(* PLC project Unnamed, Unknown Unnamed 1 *)
(* stored: creationDateTime 2025-05-12T19:02:38, modificationDateTime 2025-05-14T16:42:28 *)

PROGRAM traffic
  VAR
    pedestrianButton AT %IX0.0 : BOOL;
    systemButton0 AT %IX0.1 : BOOL;
    pR AT %QX0.4 : BOOL;
    pY AT %QX0.3 : BOOL;
    pG AT %QX0.2 : BOOL;
    cR AT %QX0.7 : BOOL;
    cY AT %QX0.6 : BOOL;
    cG AT %QX0.5 : BOOL;
  END_VAR
  VAR
    TOF0 : TOF;
    SR0 : SR;
    TOF1 : TOF;
    TOF3 : TOF;
    TOF2 : TOF;
    TOF5 : TOF;
    TOF6 : TOF;
  END_VAR
  VAR  (* added by the conversion: wires and edge detectors of the diagram *)
    R_TRIG1 : R_TRIG;
    F_TRIG2 : F_TRIG;
    F_TRIG3 : F_TRIG;
    F_TRIG4 : F_TRIG;
    R_TRIG5 : R_TRIG;
    F_TRIG6 : F_TRIG;
    R_TRIG7 : R_TRIG;
    F_TRIG8 : F_TRIG;
    F_TRIG9 : F_TRIG;
    _XOR52_OUT : BOOL;
  END_VAR

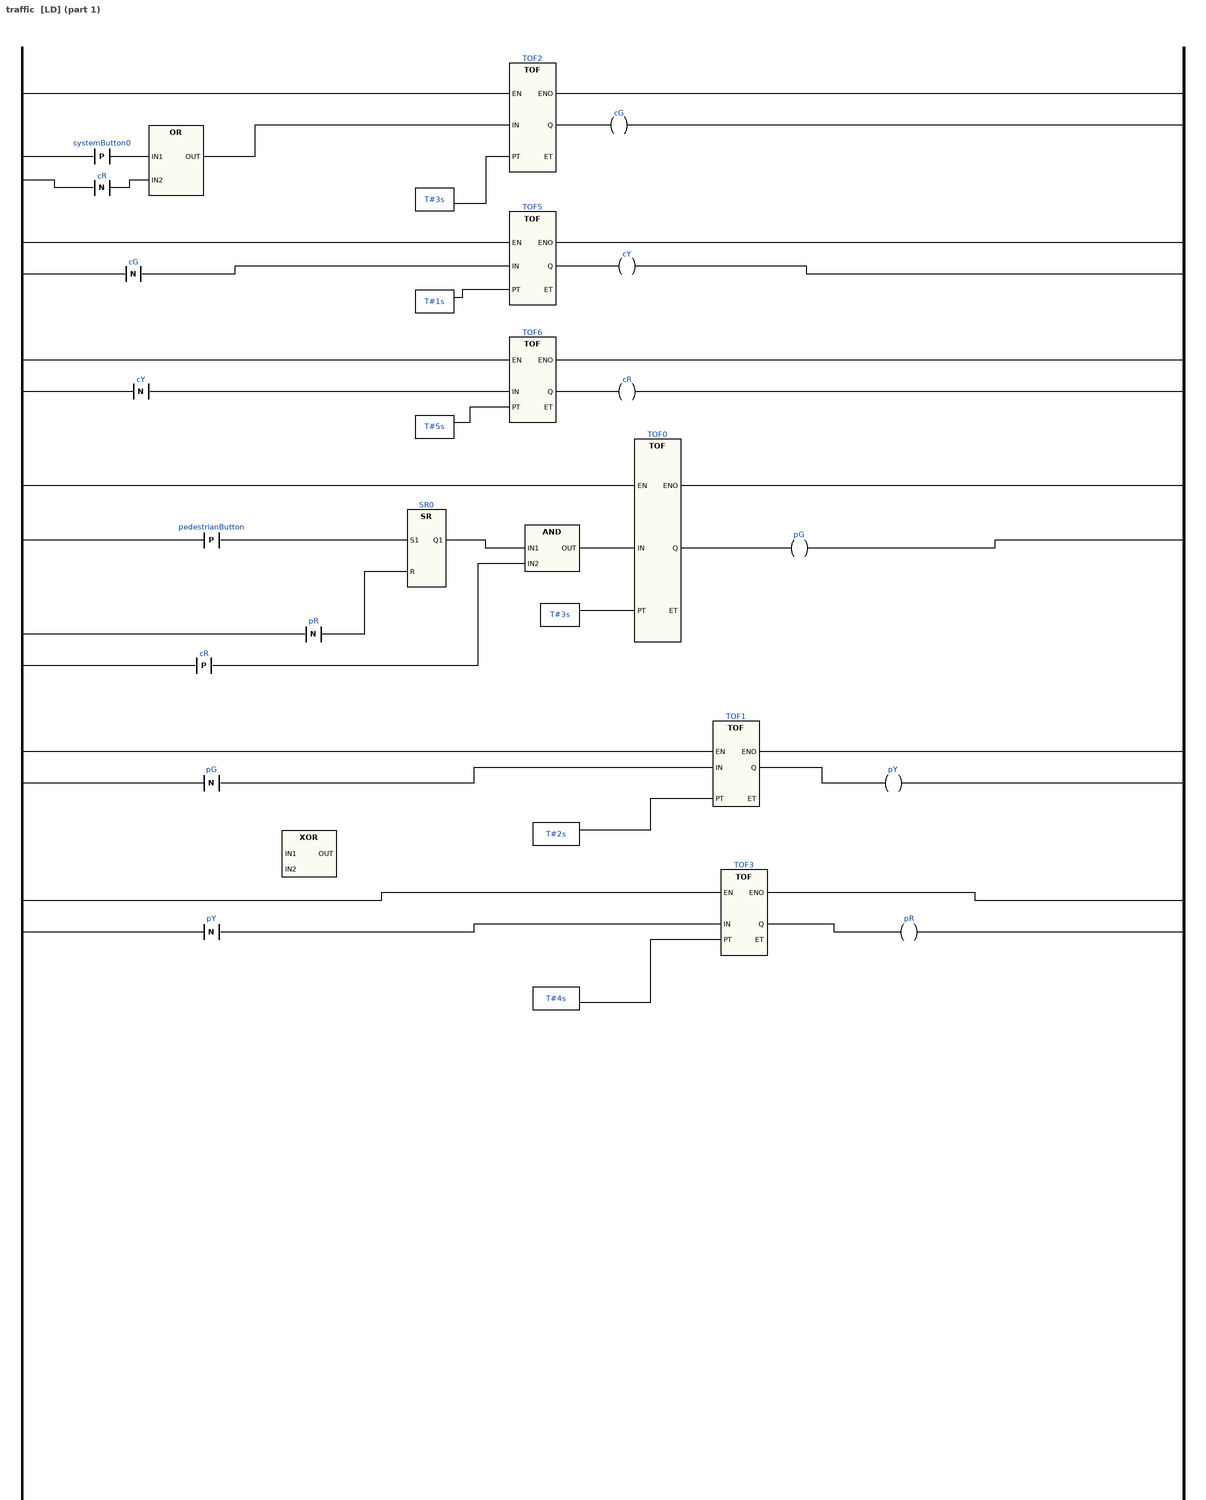
(* LD diagram, written out as Structured Text *)
R_TRIG1(CLK := systemButton0);
F_TRIG2(CLK := cR);
TOF2(IN := R_TRIG1.Q OR F_TRIG2.Q, PT := T#3s);
cG := TOF2.Q;
F_TRIG3(CLK := cG);
TOF5(IN := F_TRIG3.Q, PT := T#1s);
cY := TOF5.Q;
F_TRIG4(CLK := cY);
TOF6(IN := F_TRIG4.Q, PT := T#5s);
cR := TOF6.Q;
R_TRIG5(CLK := pedestrianButton);
F_TRIG6(CLK := pR);
SR0(S1 := R_TRIG5.Q, R := F_TRIG6.Q);
R_TRIG7(CLK := cR);
TOF0(IN := SR0.Q1 AND R_TRIG7.Q, PT := T#3s);
pG := TOF0.Q;
F_TRIG8(CLK := pG);
TOF1(IN := F_TRIG8.Q, PT := T#2s);
pY := TOF1.Q;
F_TRIG9(CLK := pY);
TOF3(IN := F_TRIG9.Q, PT := T#4s);
pR := TOF3.Q;
_XOR52_OUT := XOR();
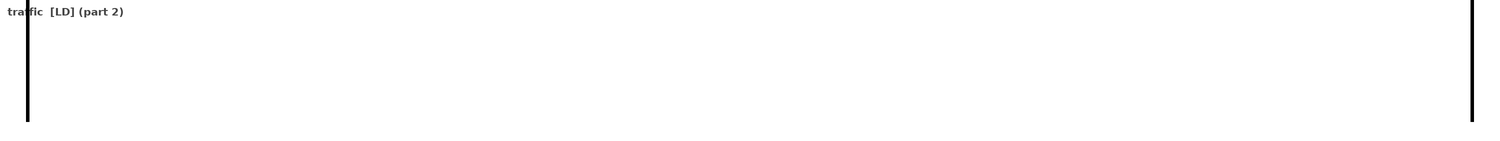
END_PROGRAM

CONFIGURATION Config0
  RESOURCE Res0 ON PLC
    TASK task0(INTERVAL := T#20ms, PRIORITY := 0);
    PROGRAM instance0 WITH task0 : traffic;
  END_RESOURCE
END_CONFIGURATION
